TYPE ST_BaseHMIConnectorEvents_ListToDisplay :
STRUCT
	arrToDisplay				: ARRAY [1..GVL_BaseConstans.MAX_EVENTS_TO_SHOW] OF ST_BaseHMIConnectorEvents_ListToDisplayRow;
	iNumberOfRow				: INT;

END_STRUCT
END_TYPE

(* stored: Version 1.1.0.1
   DUT ST_BaseHMIConnectorEvents_ListToDisplay: Id {a76f8388-425a-0985-338a-d3a600172d4b} *)
